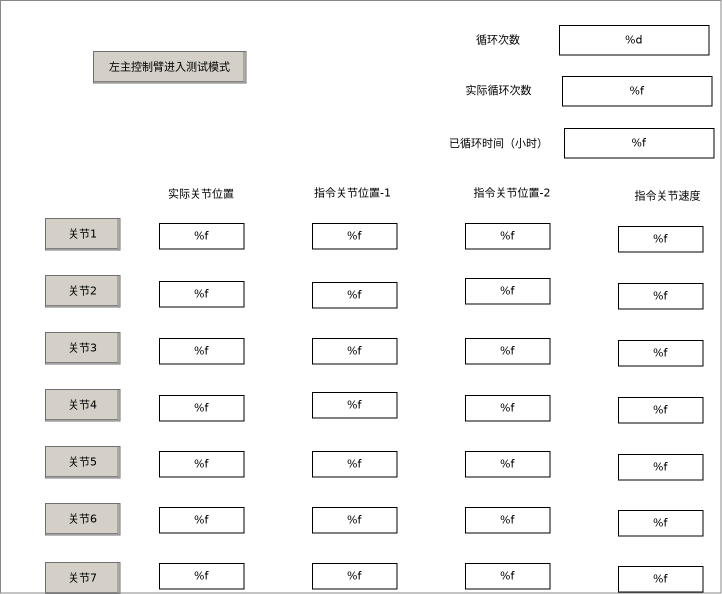
VISUALIZATION leftArmCycleTest  // 722x594
    Button (93,51 153x32), "左主控制臂进入测试模式", colour toggle: g_cycleTest.m_enterCycleTestMode[1]
        toggle g_cycleTest.m_enterCycleTestMode[1]
    Rectangle (559,25 150x30), "%d", text variable: g_cycleTest.m_targetCycleNum[1]
        OnMouseClick: write the text variable via Default
    Label (456,25 84x30), "循环次数"
    Label (293,179 119x28), "指令关节位置-1"
    Label (151,179 100x30), "实际关节位置"
    Rectangle (159,395 85x26), "%f", text variable: g_systemInfo.m_armJntInfo[1,4].m_curJntPos
    Rectangle (159,451 85x26), "%f", text variable: g_systemInfo.m_armJntInfo[1,5].m_curJntPos
    Rectangle (159,507 85x26), "%f", text variable: g_systemInfo.m_armJntInfo[1,6].m_curJntPos
    Rectangle (159,563 85x26), "%f", text variable: g_systemInfo.m_armJntInfo[1,7].m_curJntPos
    Rectangle (159,223 85x26), "%f", text variable: g_systemInfo.m_armJntInfo[1,1].m_curJntPos
    Rectangle (159,281 85x26), "%f", text variable: g_systemInfo.m_armJntInfo[1,2].m_curJntPos
    Rectangle (159,338 85x26), "%f", text variable: g_systemInfo.m_armJntInfo[1,3].m_curJntPos
    Rectangle (312,223 85x26), "%f", text variable: g_cycleTest.m_armCmdJntPos[1,1][1]
        OnMouseClick: write the text variable via Default
    Rectangle (312,282 85x26), "%f", text variable: g_cycleTest.m_armCmdJntPos[1,1][2]
        OnMouseClick: write the text variable via Default
    Rectangle (312,338 85x26), "%f", text variable: g_cycleTest.m_armCmdJntPos[1,1][3]
        OnMouseClick: write the text variable via Default
    Rectangle (312,392 85x26), "%f", text variable: g_cycleTest.m_armCmdJntPos[1,1][4]
        OnMouseClick: write the text variable via Default
    Rectangle (312,451 85x26), "%f", text variable: g_cycleTest.m_armCmdJntPos[1,1][5]
        OnMouseClick: write the text variable via Default
    Rectangle (312,507 85x26), "%f", text variable: g_cycleTest.m_armCmdJntPos[1,1][6]
        OnMouseClick: write the text variable via Default
    Rectangle (312,563 85x26), "%f", text variable: g_cycleTest.m_armCmdJntPos[1,1][7]
        OnMouseClick: write the text variable via Default
    Label (454,179 116x28), "指令关节位置-2"
    Rectangle (465,223 85x26), "%f", text variable: g_cycleTest.m_armCmdJntPos[1,2][1]
        OnMouseClick: write the text variable via Default
    Rectangle (465,278 85x26), "%f", text variable: g_cycleTest.m_armCmdJntPos[1,2][2]
        OnMouseClick: write the text variable via Default
    Rectangle (465,338 85x26), "%f", text variable: g_cycleTest.m_armCmdJntPos[1,2][3]
        OnMouseClick: write the text variable via Default
    Rectangle (465,395 85x26), "%f", text variable: g_cycleTest.m_armCmdJntPos[1,2][4]
        OnMouseClick: write the text variable via Default
    Rectangle (465,451 85x26), "%f", text variable: g_cycleTest.m_armCmdJntPos[1,2][5]
        OnMouseClick: write the text variable via Default
    Rectangle (465,507 85x26), "%f", text variable: g_cycleTest.m_armCmdJntPos[1,2][6]
        OnMouseClick: write the text variable via Default
    Rectangle (465,563 85x26), "%f", text variable: g_cycleTest.m_armCmdJntPos[1,2][7]
        OnMouseClick: write the text variable via Default
    Label (613,182 109x28), "指令关节速度"
    Rectangle (618,226 85x26), "%f", text variable: g_cycleTest.m_armCmdJntVel[1][1]
        OnMouseClick: write the text variable via Default
    Rectangle (618,283 85x26), "%f", text variable: g_cycleTest.m_armCmdJntVel[1][2]
        OnMouseClick: write the text variable via Default
    Rectangle (618,340 85x26), "%f", text variable: g_cycleTest.m_armCmdJntVel[1][3]
        OnMouseClick: write the text variable via Default
    Rectangle (618,397 85x26), "%f", text variable: g_cycleTest.m_armCmdJntVel[1][4]
        OnMouseClick: write the text variable via Default
    Rectangle (618,454 85x26), "%f", text variable: g_cycleTest.m_armCmdJntVel[1][5]
        OnMouseClick: write the text variable via Default
    Rectangle (618,510 85x26), "%f", text variable: g_cycleTest.m_armCmdJntVel[1][6]
        OnMouseClick: write the text variable via Default
    Rectangle (618,566 85x26), "%f", text variable: g_cycleTest.m_armCmdJntVel[1][7]
        OnMouseClick: write the text variable via Default
    Rectangle (562,76 150x30), "%f", text variable: g_cycleTest.m_curCycleNum[1]
        OnMouseClick: write the text variable via Default
    Label (450,80 97x21), "实际循环次数"
    Rectangle (564,128 150x30), "%f", text variable: g_cycleTest.m_curCycleTime[1]
        OnMouseClick: write the text variable via Default
    Label (438,133 121x21), "已循环时间（小时）"
    Button (45,218 75x32), "关节1", colour toggle: g_cycleTest.m_disableJntMotion[1][1]
        toggle g_cycleTest.m_disableJntMotion[1][1]
    Button (45,275 75x32), "关节2", colour toggle: g_cycleTest.m_disableJntMotion[1][2]
        toggle g_cycleTest.m_disableJntMotion[1][2]
    Button (45,332 75x32), "关节3", colour toggle: g_cycleTest.m_disableJntMotion[1][3]
        toggle g_cycleTest.m_disableJntMotion[1][3]
    Button (45,389 75x32), "关节4", colour toggle: g_cycleTest.m_disableJntMotion[1][4]
        toggle g_cycleTest.m_disableJntMotion[1][4]
    Button (45,446 75x32), "关节5", colour toggle: g_cycleTest.m_disableJntMotion[1][5]
        toggle g_cycleTest.m_disableJntMotion[1][5]
    Button (45,503 75x32), "关节6", colour toggle: g_cycleTest.m_disableJntMotion[1][6]
        toggle g_cycleTest.m_disableJntMotion[1][6]
    Button (45,562 75x32), "关节7", colour toggle: g_cycleTest.m_disableJntMotion[1][7]
        toggle g_cycleTest.m_disableJntMotion[1][7]
END_VISUALIZATION

(* stored: Version 1.1.0.1, ProductVersion 3.1.4024.11
   Visu leftArmCycleTest: Id {f69d49d0-6778-47ae-aba0-4e1dfc9c085f} *)
